// TIA Portal V18 export
DATA_BLOCK "DATA"   // DB6
{ S7_Optimized_Access := 'TRUE' }
// stored: MemoryReserve 100
   VAR
      HaveAxisStart : Bool;
      AxisStartNumber : Int;
      "Forced modification" : Bool;
   END_VAR
BEGIN
END_DATA_BLOCK
